// TIA Portal V20 export
TYPE "UDT_Service_ProcedureEnable"
   STRUCT
      Reset { ExternalAccessible := 'False'; ExternalVisible := 'False'; ExternalWritable := 'False'} : "DigValTFF";   // Reset Enablement Logic
      Start { ExternalAccessible := 'False'; ExternalVisible := 'False'; ExternalWritable := 'False'} : "DigValTFF";   // Start Enablement Logic
      Hold { ExternalAccessible := 'False'; ExternalVisible := 'False'; ExternalWritable := 'False'} : "DigValTFF";   // Hold Enablement Logic
      Unhold { ExternalAccessible := 'False'; ExternalVisible := 'False'; ExternalWritable := 'False'} : "DigValTFF";   // Unhold Enablement Logic
      Pause { ExternalAccessible := 'False'; ExternalVisible := 'False'; ExternalWritable := 'False'} : "DigValTFF";   // Pause Enablement Logic
      Resume { ExternalAccessible := 'False'; ExternalVisible := 'False'; ExternalWritable := 'False'} : "DigValTFF";   // Resume Enablement Logic
      Restart { ExternalAccessible := 'False'; ExternalVisible := 'False'; ExternalWritable := 'False'} : "DigValTFF";   // Restart Enablement Logic
      Complete { ExternalAccessible := 'False'; ExternalVisible := 'False'; ExternalWritable := 'False'} : "DigValTFF";   // Complete Enablement Logic
   END_STRUCT;
END_TYPE
